Staubli VAL3: addStrToString.pgx

public program addStrToString(string x_sInString, string& x_sOutString[], string x_sDelimiter, string& x_sSubString[])
  local num l_i
  local num l_n
begin
  // ABSTRACT:
  // This program inserts some subStrings into a specific string
  //
  // INPUT PARMS:
  //  x_sInString    : Input string into which the real values must be inserted
  //  x_sDelimiter   : Character pattern to be replaced in the input string
  //                 : Default pattern is *\../*
  //  x_sSubString[] : String value to be inserted into the input string
  //
  // OUTPUT PARMS:
  //  x_sOutString   : Output string in which subStrings have been inserted
  //
  //Created 21/12/05                              C.CURRIVAND
  //--------------------------------------------------------------
  //
  if x_sDelimiter==""
    x_sDelimiter="*\../*"
  endIf
  l_i=0
  x_sOutString=x_sInString
  l_n=find(x_sOutString,x_sDelimiter)
  while (l_i<=size(x_sSubString)-1) and (l_n!=-1)
    x_sOutString=replace(x_sOutString,x_sSubString[l_i],len(x_sDelimiter),l_n)
    l_i=l_i+1
    l_n=find(x_sOutString,x_sDelimiter)
  endWhile
end
